{attribute addProperty BoxType "EM7004-0000-9995"}
{attribute addProperty Id "OutputAT %Q*INT162"}
{attribute addProperty CRC "2526907244"}
{attribute addProperty SizeInBites "16"}
{attribute addProperty SizeInBytes "2"}
TYPE Analog_Channel_969D8B6C :
STRUCT
	{attribute addProperty Name "Output"}
	Output AT %Q* : INT;
END_STRUCT
END_TYPE

(* stored: Version 1.2.0.0, ProductVersion 3.1.4024.9
   DUT Analog_Channel_969D8B6C: Id {9f0bcd98-0935-4574-89b6-fcdc385c57b2} *)
